// TIA Portal V18 export
DATA_BLOCK "Boilers"   // DB1030
{ S7_Optimized_Access := 'FALSE' }
VERSION : 0.1
// stored: AutoNumber false, DBAccessibleFromOPCUA true, IsOnlyStoredInLoadMemory false, IsWriteProtectedInAS false
   VAR
      Boilers { S7_SetPoint := 'True'} : "UDT_BoilerUnitState";
   END_VAR
BEGIN
END_DATA_BLOCK
